{attribute 'qualified_only'}
VAR_GLOBAL
END_VAR

(* stored: Version 1.1.0.1, ProductVersion 3.1.4022.7
   GVL GVL_07_Alarm_Common: Id {cadf30b4-4410-431a-a8e1-88540b51b8a7} *)
